// TIA Portal V20 export
FUNCTION_BLOCK "FB_PartManagement"   // FB86, SCL
{ S7_Optimized_Access := 'TRUE' }
// stored: MemoryReserve 100, SetENOAutomatically false
   VAR
      sShuttle1DrilledPart : "FB_StatusPart";
      sShuttle1UndrilledPart { S7_SetPoint := 'True'} : "FB_StatusPart";
      sShuttle2DrilledPart { S7_SetPoint := 'True'} : "FB_StatusPart";
      sShuttle2UndrilledPart { S7_SetPoint := 'True'} : "FB_StatusPart";
      sShuttle1DrilledBw : "FB_StatusPart";
      sShuttle1UndrilledBw { S7_SetPoint := 'True'} : "FB_StatusPart";
      sShuttle2DrilledBw { S7_SetPoint := 'True'} : "FB_StatusPart";
      sShuttle2UndrilledBw { S7_SetPoint := 'True'} : "FB_StatusPart";
      sGripperDrilledPart : "FB_StatusPart";
      sGripperUndrilledPart { S7_SetPoint := 'True'} : "FB_StatusPart";
      sGripperDrilledBw : "FB_StatusPart";
      sGripperUndrilledBw { S7_SetPoint := 'True'} : "FB_StatusPart";
      sFixtureDrilledPart : "FB_StatusPart";
      sFixtureUndrilledPart { S7_SetPoint := 'True'} : "FB_StatusPart";
      sFixtureDrilledBw : "FB_StatusPart";
      sFixtureUndrilledBw { S7_SetPoint := 'True'} : "FB_StatusPart";
      sPosition { S7_SetPoint := 'True'} : "FB_Position";
   END_VAR
BEGIN
   REGION Description header 
       //==================================================================================
       // POSALUX Swiss SA / (C) Copyright 2026
       //----------------------------------------------------------------------------------
       // Title: FB_PartManagement
       // Comment/Function: 
       //
       // Author: Fabien WALDT
       // Engineering: TIA Portal v20
       //----------------------------------------------------------------------------------
       // Change log table:
       // Version  | Date     | Expert in charge | Changes applied
       // ---------|----------|------------------|------------------------------------
       // 00.00.01 | 20260310 | WFA              | First released version
       // ==================================================================================
   END_REGION

   REGION Shuttle 1 States
       // Drilled Part
       #sShuttle1DrilledPart(iGood := #sPosition.sShuttle1.Drilled.Presence.Part AND NOT #sShuttle1DrilledPart.iBad,
                             iUnknown := #sShuttle1DrilledPart.iUnknown,
                             iBad := #sShuttle1DrilledPart.iBad,
                             iAbsent := NOT #sPosition.sShuttle1.Drilled.Presence.Part,
                             iPresentUnexpected := "DB_LoaderShuttle1".sControlIn.sExtraPartCtrlDrilled OR "DB_LoaderShuttle1".sControlOut.sExtraPartCtrlDrilled,
                             iAbsentUnexpected := "DB_LoaderShuttle1".sControlIn.sMissingPartCtrlDrilled OR "DB_LoaderShuttle1".sControlOut.sMissingPartCtrlDrilled,
                             oStatus => #sPosition.sShuttle1.Drilled.States.Part);

       // Undrilled Part
       #sShuttle1UndrilledPart(iGood := #sPosition.sShuttle1.Undrilled.Presence.Part AND NOT #sShuttle1UndrilledPart.iBad,
                               iUnknown := #sShuttle1UndrilledPart.iUnknown,
                               iBad := #sShuttle1UndrilledPart.iBad,
                               iAbsent := NOT #sPosition.sShuttle1.Undrilled.Presence.Part,
                               iPresentUnexpected := "DB_LoaderShuttle1".sControlIn.sExtraPartCtrlUndrilled OR "DB_LoaderShuttle1".sControlOut.sExtraPartCtrlUndrilled,
                               iAbsentUnexpected := "DB_LoaderShuttle1".sControlIn.sMissingPartCtrlUndrilled OR "DB_LoaderShuttle1".sControlOut.sMissingPartCtrlUndrilled,
                               oStatus => #sPosition.sShuttle1.Undrilled.States.Part);
       // Drilled Bw
       #sShuttle1DrilledBw(iGood := #sPosition.sShuttle1.Drilled.Presence.BW AND NOT #sShuttle1DrilledBw.iBad,
                           iUnknown := #sShuttle1DrilledBw.iUnknown,
                           iBad := #sShuttle1DrilledBw.iBad,
                           iAbsent := NOT #sPosition.sShuttle1.Drilled.Presence.BW,
                           iPresentUnexpected := FALSE,
                           iAbsentUnexpected := FALSE,
                           oStatus => #sPosition.sShuttle1.Drilled.States.BW);

       // Undrilled Bw
       #sShuttle1UndrilledBw(iGood := #sPosition.sShuttle1.Undrilled.Presence.BW AND NOT #sShuttle1UndrilledBw.iBad,
                             iUnknown := #sShuttle1UndrilledBw.iUnknown,
                             iBad := #sShuttle1UndrilledBw.iBad,
                             iAbsent := NOT #sPosition.sShuttle1.Undrilled.Presence.BW,
                             iPresentUnexpected := "DB_LoaderShuttle1".sBwControlIn.sExtraBwCtrl,
                             iAbsentUnexpected := "DB_LoaderShuttle1".sBwControlIn.sMissingBwCtrl,
                             oStatus => #sPosition.sShuttle1.Undrilled.States.BW);
   END_REGION

   REGION Shuttle 2 States
       // Drilled Part
       #sShuttle2DrilledPart(iGood := #sPosition.sShuttle2.Drilled.Presence.Part AND NOT #sShuttle2DrilledPart.iBad,
                             iUnknown := #sShuttle2DrilledPart.iUnknown,
                             iBad := #sShuttle2DrilledPart.iBad,
                             iAbsent := NOT #sPosition.sShuttle2.Drilled.Presence.Part,
                             iPresentUnexpected := "DB_LoaderShuttle2".sControlIn.sExtraPartCtrlDrilled OR "DB_LoaderShuttle2".sControlOut.sExtraPartCtrlDrilled,
                             iAbsentUnexpected := "DB_LoaderShuttle2".sControlIn.sMissingPartCtrlDrilled OR "DB_LoaderShuttle2".sControlOut.sMissingPartCtrlDrilled,
                             oStatus => #sPosition.sShuttle2.Drilled.States.Part);

       // Undrilled Part
       #sShuttle2UndrilledPart(iGood := #sPosition.sShuttle2.Undrilled.Presence.Part AND NOT #sShuttle2UndrilledPart.iBad,
                               iUnknown := #sShuttle2UndrilledPart.iUnknown,
                               iBad := #sShuttle2UndrilledPart.iBad,
                               iAbsent := NOT #sPosition.sShuttle2.Undrilled.Presence.Part,
                               iPresentUnexpected := "DB_LoaderShuttle2".sControlIn.sExtraPartCtrlUndrilled OR "DB_LoaderShuttle2".sControlOut.sExtraPartCtrlUndrilled,
                               iAbsentUnexpected := "DB_LoaderShuttle2".sControlIn.sMissingPartCtrlUndrilled OR "DB_LoaderShuttle2".sControlOut.sMissingPartCtrlUndrilled,
                               oStatus => #sPosition.sShuttle2.Undrilled.States.Part);
       // Drilled Bw
       #sShuttle2DrilledBw(iGood := #sPosition.sShuttle2.Drilled.Presence.BW AND NOT #sShuttle2DrilledBw.iBad,
                           iUnknown := #sShuttle2DrilledBw.iUnknown,
                           iBad := #sShuttle2DrilledBw.iBad,
                           iAbsent := NOT #sPosition.sShuttle2.Drilled.Presence.BW,
                           iPresentUnexpected := FALSE,
                           iAbsentUnexpected := FALSE,
                           oStatus => #sPosition.sShuttle2.Drilled.States.BW);

       // Undrilled Bw
       #sShuttle2UndrilledBw(iGood := #sPosition.sShuttle2.Undrilled.Presence.BW AND NOT #sShuttle2UndrilledBw.iBad,
                             iUnknown := #sShuttle2UndrilledBw.iUnknown,
                             iBad := #sShuttle2UndrilledBw.iBad,
                             iAbsent := NOT #sPosition.sShuttle2.Undrilled.Presence.BW,
                             iPresentUnexpected := "DB_LoaderShuttle2".sBwControlIn.sExtraBwCtrl,
                             iAbsentUnexpected := "DB_LoaderShuttle2".sBwControlIn.sMissingBwCtrl,
                             oStatus => #sPosition.sShuttle2.Undrilled.States.BW);
   END_REGION

   REGION Gripper States
       // Drilled Part
       #sGripperDrilledPart(iGood := #sPosition.sGripper.Drilled.Presence.Part AND NOT #sGripperDrilledPart.iBad,
                            iUnknown := #sGripperDrilledPart.iUnknown,
                            iBad := #sGripperDrilledPart.iBad,
                            iAbsent := NOT #sPosition.sGripper.Drilled.Presence.Part,
                            iPresentUnexpected := "DB_ExtraMissingPart".sExtraPartDrilledGripper,
                            iAbsentUnexpected := "DB_ExtraMissingPart".sMissingPartDrilledGripper,
                            oStatus => #sPosition.sGripper.Drilled.States.Part);

       // Undrilled Part
       #sGripperUndrilledPart(iGood := #sPosition.sGripper.Undrilled.Presence.Part AND NOT #sGripperUndrilledPart.iBad,
                              iUnknown := #sGripperUndrilledPart.iUnknown,
                              iBad := #sGripperUndrilledPart.iBad,
                              iAbsent := NOT #sPosition.sGripper.Undrilled.Presence.Part,
                              iPresentUnexpected := "DB_ExtraMissingPart".sExtraPartUndrilledGripper,
                              iAbsentUnexpected := "DB_ExtraMissingPart".sMissingPartUndrilledGripper,
                              oStatus => #sPosition.sGripper.Undrilled.States.Part);
       // Drilled Bw
       #sGripperDrilledBw(iGood := #sPosition.sGripper.Drilled.Presence.BW AND NOT #sGripperDrilledBw.iBad,
                          iUnknown := #sGripperDrilledBw.iUnknown,
                          iBad := #sGripperDrilledBw.iBad,
                          iAbsent := NOT #sPosition.sGripper.Drilled.Presence.BW,
                          iPresentUnexpected := "DB_ExtraMissingPart".sExtraPartDrilledGripper,
                          iAbsentUnexpected := "DB_ExtraMissingPart".sMissingPartDrilledGripper,
                          oStatus => #sPosition.sGripper.Drilled.States.BW);

       // Undrilled Bw
       #sGripperUndrilledBw(iGood := #sPosition.sGripper.Undrilled.Presence.BW AND NOT #sGripperUndrilledBw.iBad,
                            iUnknown := #sGripperUndrilledBw.iUnknown,
                            iBad := #sGripperUndrilledBw.iBad,
                            iAbsent := NOT #sPosition.sGripper.Undrilled.Presence.BW,
                            iPresentUnexpected := "DB_ExtraMissingPart".sExtraPartUndrilledGripper,
                            iAbsentUnexpected := "DB_ExtraMissingPart".sMissingPartUndrilledGripper,
                            oStatus => #sPosition.sGripper.Undrilled.States.BW);
   END_REGION

   REGION Fixture States
       // Drilled - Part
       #sFixtureDrilledPart(iGood := #sPosition.sFixture.Drilled.Presence.Part AND NOT #sFixtureDrilledPart.iBad,
                            iUnknown := #sFixtureDrilledPart.iUnknown,
                            iBad := "DB_ScannerComm".oBadPart,
                            iAbsent := NOT #sPosition.sFixture.Drilled.Presence.Part AND NOT #sPosition.sFixture.Undrilled.Presence.Part,
                            iPresentUnexpected := "DB_ExtraMissingPart".sExtraPartFixture,
                            iAbsentUnexpected := "DB_ExtraMissingPart".sMissingPartFixture,
                            oStatus => #sPosition.sFixture.Drilled.States.Part);

        // Undrilled Part
       #sFixtureUndrilledPart(iGood := #sPosition.sFixture.Undrilled.Presence.Part,
                              iUnknown := #sFixtureUndrilledPart.iUnknown,
                              iBad := #sFixtureUndrilledPart.iBad,
                              iAbsent := NOT #sPosition.sFixture.Undrilled.Presence.Part,
                              iPresentUnexpected := "DB_ExtraMissingPart".sExtraPartFixture,
                              iAbsentUnexpected := "DB_ExtraMissingPart".sMissingPartFixture,
                              oStatus => #sPosition.sFixture.Undrilled.States.Part);
       // Drilled Bw 
         #sFixtureDrilledBw(iGood := (#sPosition.sFixture.Drilled.Presence.BW OR #sPosition.sFixture.Undrilled.Presence.BW) AND NOT #sGripperDrilledBw.iBad,
                            iUnknown := #sFixtureDrilledBw.iUnknown,
                            iBad := #sFixtureDrilledBw.iBad,
                            iAbsent := NOT #sPosition.sFixture.Drilled.Presence.BW AND NOT #sPosition.sFixture.Undrilled.Presence.BW,
                            iPresentUnexpected := "DB_ExtraMissingPart".sExtraPartFixture,
                            iAbsentUnexpected := "DB_ExtraMissingPart".sMissingPartFixture,
                            oStatus => #sPosition.sFixture.Drilled.States.BW);

       // Undrilled Bw
       #sGripperUndrilledBw(iGood := #sPosition.sFixture.Undrilled.Presence.BW,
                            iUnknown := #sGripperUndrilledBw.iUnknown,
                            iBad := #sGripperUndrilledBw.iBad,
                            iAbsent := NOT #sPosition.sFixture.Undrilled.Presence.BW,
                            iPresentUnexpected := "DB_ExtraMissingPart".sExtraPartFixture,
                            iAbsentUnexpected := "DB_ExtraMissingPart".sMissingPartFixture,
                            oStatus => #sPosition.sFixture.Undrilled.States.BW);
   END_REGION

   REGION Position
       #sPosition(iCondPartInSh1 := (("DB_LoaderShuttle1".sExtLoadUnload.sCurrent_Step_NB = 60 OR "DB_LoaderShuttle1".sExtLoadUnload.sCurrent_Step_NB = 120) AND NOT "DB_WorkingModes".sEmptying),
                  iCondBwInSh1 := "DB_LoaderShuttle1".sBwLoadUnload.sInterface.JobDone AND "DB_LoaderShuttle1".sBwLoadUnload.iLoadReq,
                  iCondPartInSh2 := (("DB_LoaderShuttle2".sExtLoadUnload.sCurrent_Step_NB = 60 OR "DB_LoaderShuttle2".sExtLoadUnload.sCurrent_Step_NB = 120) AND NOT "DB_WorkingModes".sEmptying),
                  iCondBwInSh2 := "DB_LoaderShuttle2".sBwLoadUnload.sInterface.JobDone AND "DB_LoaderShuttle2".sBwLoadUnload.iLoadReq,
                  iCondPartPresCtrlInSh1 := "DB_LoaderShuttle1".sControlIn.sCurrent_Step_NB = 140 AND NOT "DB_WorkingModes".sEmptying,
                  iCondBWPresCtrlInSh1 := "DB_LoaderShuttle1".sBwControlIn.sCurrent_Step_NB = 40,
                  iCondPartPresCtrlInSh2 := "DB_LoaderShuttle2".sControlIn.sCurrent_Step_NB = 140,
                  iCondBWPresCtrlInSh2 := "DB_LoaderShuttle2".sBwControlIn.sCurrent_Step_NB = 40,
                  iCondPartPresCtrlOutSh1 := "DB_LoaderShuttle1".sControlOut.sCurrent_Step_NB = 140,
                  iCondPartPresCtrlOutSh2 := "DB_LoaderShuttle2".sControlOut.sCurrent_Step_NB = 140,
                  iUndrilledPartPresence := "DB_DigitalInputsBW_Station".sUndrilledPartCtrl.sSWStatus,
                  iDrilledPartPresence := "DB_DigitalInputsBW_Station".sDrilledPartCtrl.sSWStatus,
                  iUndrilledBWPresence := "DB_DigitalInputsBW_Station".sBwCtrl.sSWStatus,
                  iCloseReqLoadGripperSh1 := "DB_LoaderShuttle1".sIntLoadUnload.oLoadGripperCloseReq OR "DB_LoaderShuttle1".sIntLoadUnloadOP.oLoadGripperCloseReq,
                  iCloseReqLoadGripperSh2 := "DB_LoaderShuttle2".sIntLoadUnload.oLoadGripperCloseReq OR "DB_LoaderShuttle2".sIntLoadUnloadOP.oLoadGripperCloseReq,
                  iCloseReqFixture := "DB_GestionFixture".sFixtureHold,
                  iDrilling_Finished := "DB_ScannerComm".oEndOfJob OR #sPosition.iDrilling_Finished,
                  iCloseReqUnloadGripper := "DB_GestionGripper".sUnloadGripperCloseReq,
                  iOpenReqUnloadGripperSh1 := "DB_LoaderShuttle1".sIntLoadUnload.oUnloadGripperOpenReq OR "DB_LoaderShuttle1".sIntLoadUnloadOP.oUnloadGripperOpenReq,
                  iOpenReqUnloadGripperSh2 := "DB_LoaderShuttle2".sIntLoadUnload.oUnloadGripperOpenReq OR "DB_LoaderShuttle2".sIntLoadUnloadOP.oUnloadGripperOpenReq,
                  iCondPartOutSh1 := (("DB_LoaderShuttle1".sExtLoadUnload.sInterface.JobDone AND NOT "DB_WorkingModes".sFilling) AND NOT "DB_WorkingModes".sSemiAuto) OR ( "DB_LoaderShuttle1".sExtLoadUnload.sCurrent_Step_NB = 150 AND "DB_WorkingModes".sSemiAuto),
                  iCondBwOutSh1 := "DB_LoaderShuttle1".sBwLoadUnload.sInterface.JobDone AND "DB_LoaderShuttle1".sBwLoadUnload.iUnloadReq,
                  iCondPartOutSh2 := (("DB_LoaderShuttle2".sExtLoadUnload.sInterface.JobDone AND NOT "DB_WorkingModes".sFilling) AND NOT "DB_WorkingModes".sSemiAuto) OR ( "DB_LoaderShuttle2".sExtLoadUnload.sCurrent_Step_NB = 150 AND "DB_WorkingModes".sSemiAuto),
                  iCondBwOutSh2 := "DB_LoaderShuttle2".sBwLoadUnload.sInterface.JobDone AND "DB_LoaderShuttle2".sBwLoadUnload.iUnloadReq);
   END_REGION
END_FUNCTION_BLOCK
